{attribute 'reflection'} 
FUNCTION_BLOCK FB_Logger
VAR_INPUT
	iLogging:			I_Logging;
END_VAR
VAR_OUTPUT
	fbArguments:				FB_Argument;
END_VAR
VAR
    {attribute 'hide'} 
    {attribute 'instance-path'} 
    {attribute 'noinit'} 
    sInstancePath:				STRING(255); 
END_VAR

//FB_Init ist immer implizit verfügbar und wird primär für die Initialisierung verwendet.
//Der Rückgabewert wird nicht ausgewertet. Für gezielte Einflussnahme können Sie
//die Methoden explizit deklarieren und darin mit dem Standard-Initialisierungscode 
//zusätzlichen Code bereitstellen. Sie können den Rückgabewert auswerten.
METHOD FB_Init: BOOL
VAR_INPUT    
bInitRetains: BOOL; // TRUE: Die Retain-Variablen werden initialisiert (Reset warm / Reset kalt)    
bInCopyCode: BOOL;  // TRUE: Die Instanz wird danach in den Kopiercode kopiert (Online-Change)
END_VAR
sInstancePath:= F_InstancePath(sInstancePath);
END_METHOD

METHOD PUBLIC M_Critical : BOOL
VAR_INPUT
	nID:				UDINT;
	sMessage:			STRING(255);
END_VAR
VAR
	stMessage:			ST_Message;
END_VAR
IF iLogging = 0 THEN
	RETURN;
END_IF

stMessage.eLogLevel:= E_LogLevel.Critical;
stMessage.nID:= nID;
stMessage.nTimestamp:= F_GetSystemTime();
stMessage.sMessage:= sMessage;
stMessage.sArguments:= fbArguments.P_Value;
stMessage.sDefault:= F_Format(sMessage, fbArguments.P_Value);
stMessage.sSource:= sInstancePath;
fbArguments.M_Clear();

iLogging.M_Log(stMessage);
END_METHOD

METHOD PUBLIC M_Error : BOOL
VAR_INPUT
	nID:				UDINT;
	sMessage:			STRING(255);
END_VAR
VAR
	stMessage:			ST_Message;
END_VAR
IF iLogging = 0 THEN
	RETURN;
END_IF

stMessage.eLogLevel:= E_LogLevel.Error;
stMessage.nID:= nID;
stMessage.nTimestamp:= F_GetSystemTime();
stMessage.sMessage:= sMessage;
stMessage.sArguments:= fbArguments.P_Value;
stMessage.sDefault:= F_Format(sMessage, fbArguments.P_Value);
stMessage.sSource:= sInstancePath;
fbArguments.M_Clear();

iLogging.M_Log(stMessage);
END_METHOD

METHOD PUBLIC M_Info : BOOL
VAR_INPUT
	nID:				UDINT;
	sMessage:			STRING(255);
END_VAR
VAR
	stMessage:			ST_Message;
END_VAR
IF iLogging = 0 THEN
	RETURN;
END_IF

stMessage.eLogLevel:= E_LogLevel.Info;
stMessage.nID:= nID;
stMessage.nTimestamp:= F_GetSystemTime();
stMessage.sMessage:= sMessage;
stMessage.sArguments:= fbArguments.P_Value;
stMessage.sDefault:= F_Format(sMessage, fbArguments.P_Value);
stMessage.sSource:= sInstancePath;
fbArguments.M_Clear();

iLogging.M_Log(stMessage);
END_METHOD

METHOD PUBLIC M_Verbose : BOOL
VAR_INPUT
	sMessage:			STRING(255);
END_VAR
VAR
	stMessage:			ST_Message;
END_VAR
IF iLogging = 0 THEN
	RETURN;
END_IF

stMessage.eLogLevel:= E_LogLevel.Verbose;
stMessage.nID:= 0;
stMessage.nTimestamp:= F_GetSystemTime();
stMessage.sMessage:= sMessage;
stMessage.sArguments:= fbArguments.P_Value;
stMessage.sDefault:= F_Format(sMessage, fbArguments.P_Value);
stMessage.sSource:= sInstancePath;
fbArguments.M_Clear();

iLogging.M_Log(stMessage);
END_METHOD

METHOD PUBLIC M_Warning : BOOL
VAR_INPUT
	nID:				UDINT;
	sMessage:			STRING(255);
END_VAR
VAR
	stMessage:			ST_Message;
END_VAR
IF iLogging = 0 THEN
	RETURN;
END_IF

stMessage.eLogLevel:= E_LogLevel.Warning;
stMessage.nID:= nID;
stMessage.nTimestamp:= F_GetSystemTime();
stMessage.sMessage:= sMessage;
stMessage.sArguments:= fbArguments.P_Value;
stMessage.sDefault:= F_Format(sMessage, fbArguments.P_Value);
stMessage.sSource:= sInstancePath;
fbArguments.M_Clear();

iLogging.M_Log(stMessage);
END_METHOD

PROPERTY PUBLIC P_Argument : I_Argument
GET
P_Argument:= fbArguments;
END_GET
END_PROPERTY

PROPERTY PUBLIC P_Logger : I_Logging
GET
P_Logger:= iLogging;
END_GET
SET
iLogging:= P_Logger;
END_SET
END_PROPERTY

END_FUNCTION_BLOCK

(* stored: Version 1.1.0.1
   POU FB_Logger: Id {fcfa56ff-d0f1-4149-9de7-6f44354915c6}, SpecialFunc None
   Method FB_Init: Id {256fe292-0b03-4593-83b5-0da540634dee}
   Method M_Critical: Id {7b4c91bf-8e3c-413c-a148-e271617106d9}
   Method M_Error: Id {11687e23-ea95-4e4f-aed4-4799ffa1ad84}
   Method M_Info: Id {7a920e55-da6d-473b-9aba-119c4de007e0}
   Method M_Verbose: Id {db95e385-16ed-493b-a6a5-28cc6625776b}
   Method M_Warning: Id {1aa0d3ef-0f74-4102-97d7-7d587822db85}
   Property P_Argument: Id {dd3bce54-33d7-4a6c-8d06-ad6a5d0ec566}
   Get Get: Id {9148b4be-b1fa-4fe4-a389-e96c939bba14}
   Property P_Logger: Id {98c079df-4944-4aae-a3d6-ca12ac41d1d4}
   Get Get: Id {7f49254e-94b6-4972-a1b5-02a92d10e780}
   Set Set: Id {4bbb606c-4053-49cc-ae04-84e1809ace25} *)
